Staubli VAL3: setYaxis.pgx

program setYaxis()
begin
  numMessage[4]=0
  //-------------------------------set carrier to default
  stringYarray=""
  while numMessage[4]==0
    sioGet(sioASCII,numMessage)
    stringYarray=chr(numMessage[0])
    if chr(numMessage[1])!="#"
      stringYarray=stringYarray+chr(numMessage[1])
      //stringYarray=chr(numMessage[4])
    endIf
    toNum(stringYarray,numYarray,isNum)
    putln(stringYarray)
  endWhile
end
